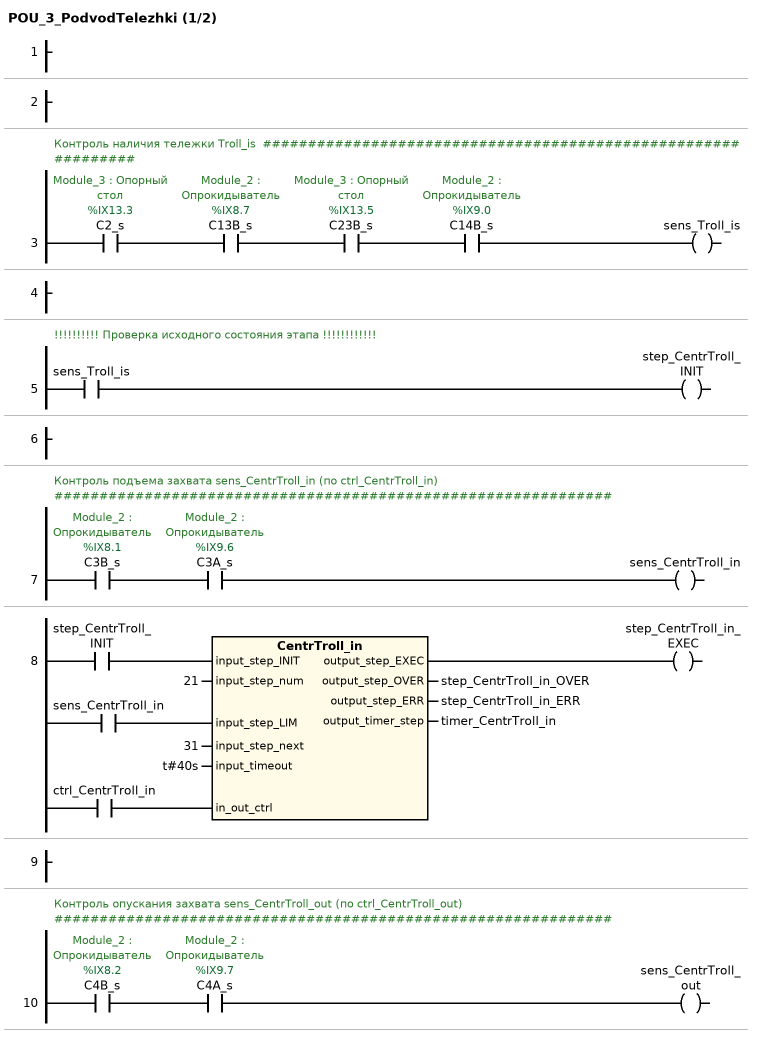
// NETWORK 1

// NETWORK 2

// NETWORK 3
// Контроль наличия тележки Troll_is  ##############################################################
//   C2_s: Module_3 : Опорный стол | AT %IX13.3
//   C13B_s: Module_2 : Опрокидыватель | AT %IX8.7
//   C23B_s: Module_3 : Опорный стол | AT %IX13.5
//   C14B_s: Module_2 : Опрокидыватель | AT %IX9.0
sens_Troll_is := C2_s AND C13B_s AND C23B_s AND C14B_s;

// NETWORK 4

// NETWORK 5
// !!!!!!!!!! Проверка исходного состояния этапа !!!!!!!!!!!!
step_CentrTroll_INIT := sens_Troll_is;

// NETWORK 6

// NETWORK 7
// Контроль подъема захвата sens_CentrTroll_in (по ctrl_CentrTroll_in) ##############################################################
//   C3B_s: Module_2 : Опрокидыватель | AT %IX8.1
//   C3A_s: Module_2 : Опрокидыватель | AT %IX9.6
sens_CentrTroll_in := C3B_s AND C3A_s;

// NETWORK 8
CentrTroll_in(input_step_INIT := step_CentrTroll_INIT, input_step_num := 21, input_step_LIM := sens_CentrTroll_in, input_step_next := 31, input_timeout := t#40s, in_out_ctrl := ctrl_CentrTroll_in, output_step_OVER => step_CentrTroll_in_OVER, output_step_ERR => step_CentrTroll_in_ERR, output_timer_step => timer_CentrTroll_in);
step_CentrTroll_in_EXEC := CentrTroll_in.output_step_EXEC;

// NETWORK 9

// NETWORK 10
// Контроль опускания захвата sens_CentrTroll_out (по ctrl_CentrTroll_out) ##############################################################
//   C4B_s: Module_2 : Опрокидыватель | AT %IX8.2
//   C4A_s: Module_2 : Опрокидыватель | AT %IX9.7
sens_CentrTroll_out := C4B_s AND C4A_s;

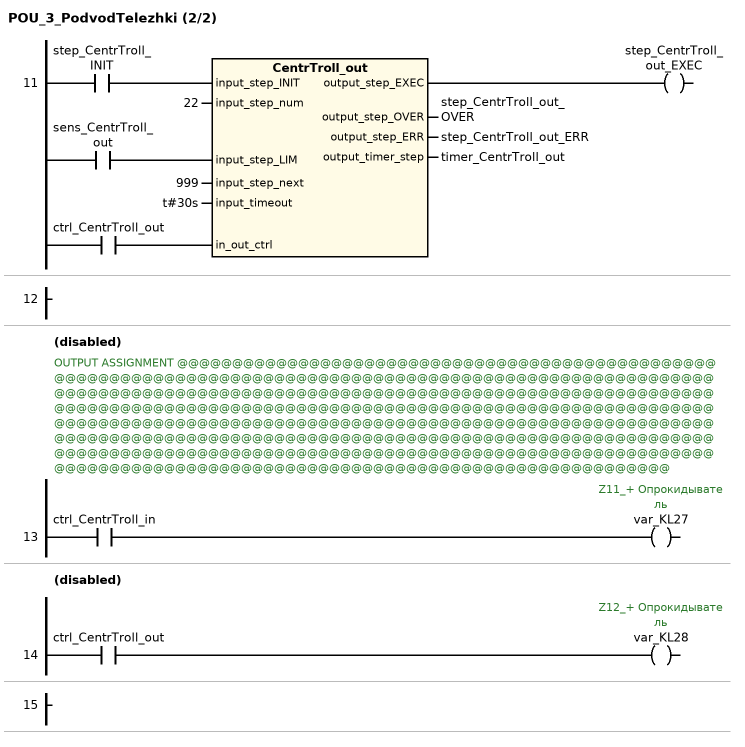
// NETWORK 11
CentrTroll_out(input_step_INIT := step_CentrTroll_INIT, input_step_num := 22, input_step_LIM := sens_CentrTroll_out, input_step_next := 999, input_timeout := t#30s, in_out_ctrl := ctrl_CentrTroll_out, output_step_OVER => step_CentrTroll_out_OVER, output_step_ERR => step_CentrTroll_out_ERR, output_timer_step => timer_CentrTroll_out);
step_CentrTroll_out_EXEC := CentrTroll_out.output_step_EXEC;

// NETWORK 12

// NETWORK 13 (disabled)
// OUTPUT ASSIGNMENT @@@@@@@@@@@@@@@@@@@@@@@@@@@@@@@@@@@@@@@@@@@@@@@@@@@@@@@@@@@@@@@@@@@@@@@@@@@@@@@@@@@@@@@@@@@@@@@@@@@@@@@@@@@@@@@@@@@@@@@@@@@@@@@@@@@@@@@@@@@@@@@@@@@@@@@@@@@@@@@@@@@@@@@@@@@@@@@@@@@@@@@@@@@@@@@@@@@@@@@@@@@@@@@@@@@@@@@@@@@@@@@@@@@@@@@@@@@@@@@@@@@@@@@@@@@@@@@@@@@@@@@@@@@@@@@@@@@@@@@@@@@@@@@@@@@@@@@@@@@@@@@@@@@@@@@@@@@@@@@@@@@@@@@@@@@@@@@@@@@@@@@@@@@@@@@@@@@@@@@@@@@@@@@@@@@@@@@@@@@@@@@@@@@@@@@@@@@@@@@@@@@@@@@@@@@@@@@@@@@@@@@@@@@@@@@@@@@@@@@@@@@@@@@@@@@@@@@@@@@@@@@@@
//   var_KL27: Z11_+ Опрокидыватель
// var_KL27 := ctrl_CentrTroll_in;

// NETWORK 14 (disabled)
//   var_KL28: Z12_+ Опрокидыватель
// var_KL28 := ctrl_CentrTroll_out;

// NETWORK 15

END_PROGRAM

// MyController/Application/module_unites/CentrTroll_in
PROGRAM CentrTroll_in
VAR_INPUT
	input_step_INIT: BOOL;
	input_step_num: INT;
	input_step_LIM: BOOL;
	input_step_next: INT;
	input_timeout: TIME;
END_VAR

VAR_OUTPUT
	output_step_EXEC: BOOL;
	output_step_OVER: BOOL;
	output_step_ERR: BOOL;
	output_timer_step: TIME;
END_VAR
VAR_IN_OUT
	in_out_ctrl: BOOL;
END_VAR
VAR
	TON_step: TON;
	TON_step_res: BOOL;
	step_active: BOOL;
	TON_delay: TON;
	timer_delay: TIME;
	ton_delay_ok: BOOL;
END_VAR
VAR // added by the converter: edge detectors and wires of the graphical bodies
    _rt1, _rt2, _rt3, _rt4, _rt5, _rt6, _rt7 : R_TRIG;
    _w1, _w2 : BOOL;
    _ft1 : F_TRIG;
END_VAR

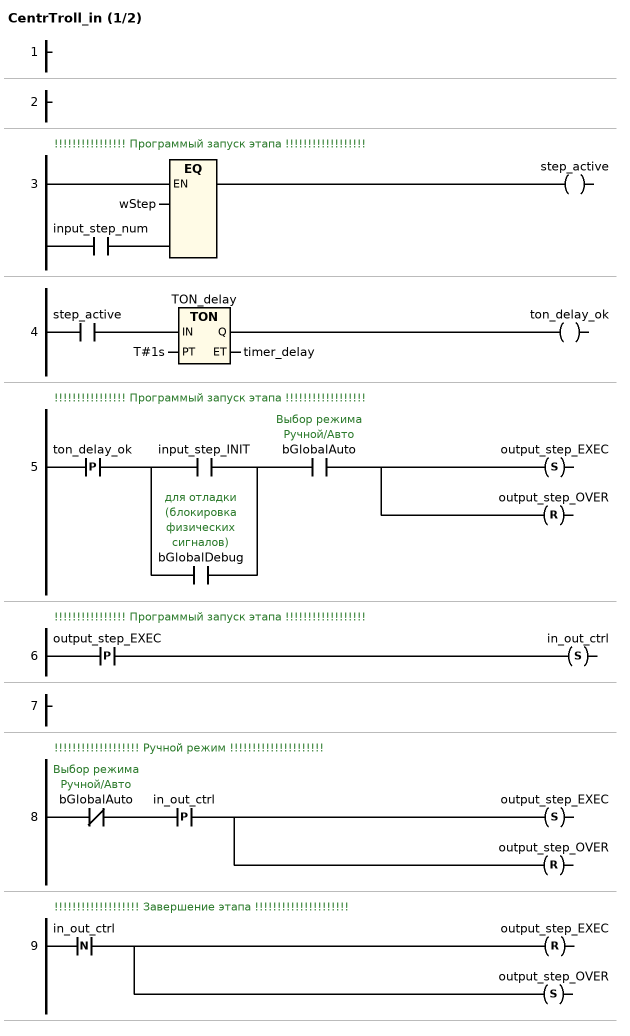
// NETWORK 1

// NETWORK 2

// NETWORK 3
// !!!!!!!!!!!!!!!! Программый запуск этапа !!!!!!!!!!!!!!!!!!
step_active := wStep = input_step_num;

// NETWORK 4
TON_delay(IN := step_active, PT := T#1s, ET => timer_delay); // TON
ton_delay_ok := TON_delay.Q;

// NETWORK 5
// !!!!!!!!!!!!!!!! Программый запуск этапа !!!!!!!!!!!!!!!!!!
//   bGlobalDebug: для отладки (блокировка физических сигналов)
//   bGlobalAuto: Выбор режима Ручной/Авто
_rt1(CLK := ton_delay_ok);
_w1 := _rt1.Q AND (input_step_INIT OR bGlobalDebug) AND bGlobalAuto;
output_step_EXEC S= _w1;
output_step_OVER R= _w1;

// NETWORK 6
// !!!!!!!!!!!!!!!! Программый запуск этапа !!!!!!!!!!!!!!!!!!
_rt2(CLK := output_step_EXEC);
in_out_ctrl S= _rt2.Q;

// NETWORK 7

// NETWORK 8
// !!!!!!!!!!!!!!!!!!! Ручной режим !!!!!!!!!!!!!!!!!!!!!
//   bGlobalAuto: Выбор режима Ручной/Авто
_rt3(CLK := in_out_ctrl);
_w2 := NOT bGlobalAuto AND _rt3.Q;
output_step_EXEC S= _w2;
output_step_OVER R= _w2;

// NETWORK 9
// !!!!!!!!!!!!!!!!!!! Завершение этапа !!!!!!!!!!!!!!!!!!!!!
_ft1(CLK := in_out_ctrl);
output_step_EXEC R= _ft1.Q;
output_step_OVER S= _ft1.Q;

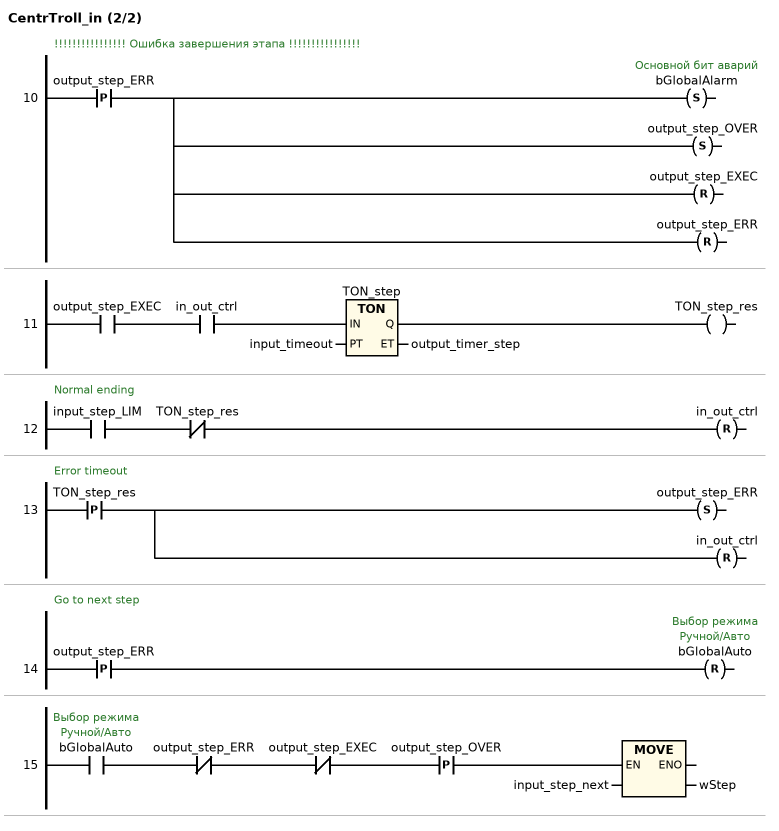
// NETWORK 10
// !!!!!!!!!!!!!!!! Ошибка завершения этапа !!!!!!!!!!!!!!!!
//   bGlobalAlarm: Основной бит аварий
_rt4(CLK := output_step_ERR);
bGlobalAlarm S= _rt4.Q;
output_step_OVER S= _rt4.Q;
output_step_EXEC R= _rt4.Q;
output_step_ERR R= _rt4.Q;

// NETWORK 11
TON_step(IN := output_step_EXEC AND in_out_ctrl, PT := input_timeout, ET => output_timer_step); // TON
TON_step_res := TON_step.Q;

// NETWORK 12
// Normal ending
in_out_ctrl R= input_step_LIM AND NOT TON_step_res;

// NETWORK 13
// Error timeout
_rt5(CLK := TON_step_res);
output_step_ERR S= _rt5.Q;
in_out_ctrl R= _rt5.Q;

// NETWORK 14
// Go to next step
//   bGlobalAuto: Выбор режима Ручной/Авто
_rt6(CLK := output_step_ERR);
bGlobalAuto R= _rt6.Q;

// NETWORK 15
//   bGlobalAuto: Выбор режима Ручной/Авто
_rt7(CLK := output_step_OVER);
IF bGlobalAuto AND NOT output_step_ERR AND NOT output_step_EXEC AND _rt7.Q THEN wStep := input_step_next; END_IF

END_PROGRAM

// MyController/Application/module_unites/CentrTroll_out
PROGRAM CentrTroll_out
VAR_INPUT
	input_step_INIT: BOOL;
	input_step_num: INT;
	input_step_LIM: BOOL;
	input_step_next: INT;
	input_timeout: TIME;
END_VAR

VAR_OUTPUT
	output_step_EXEC: BOOL;
	output_step_OVER: BOOL;
	output_step_ERR: BOOL;
	output_timer_step: TIME;
END_VAR
VAR_IN_OUT
	in_out_ctrl: BOOL;
END_VAR
VAR
	TON_step: TON;
	TON_step_res: BOOL;
	step_active: BOOL;
	TON_delay: TON;
	timer_delay: TIME;
	ton_delay_ok: BOOL;
END_VAR
VAR // added by the converter: edge detectors and wires of the graphical bodies
    _rt1, _rt2, _rt3, _rt4, _rt5, _rt6, _rt7 : R_TRIG;
    _w1, _w2 : BOOL;
    _ft1 : F_TRIG;
END_VAR

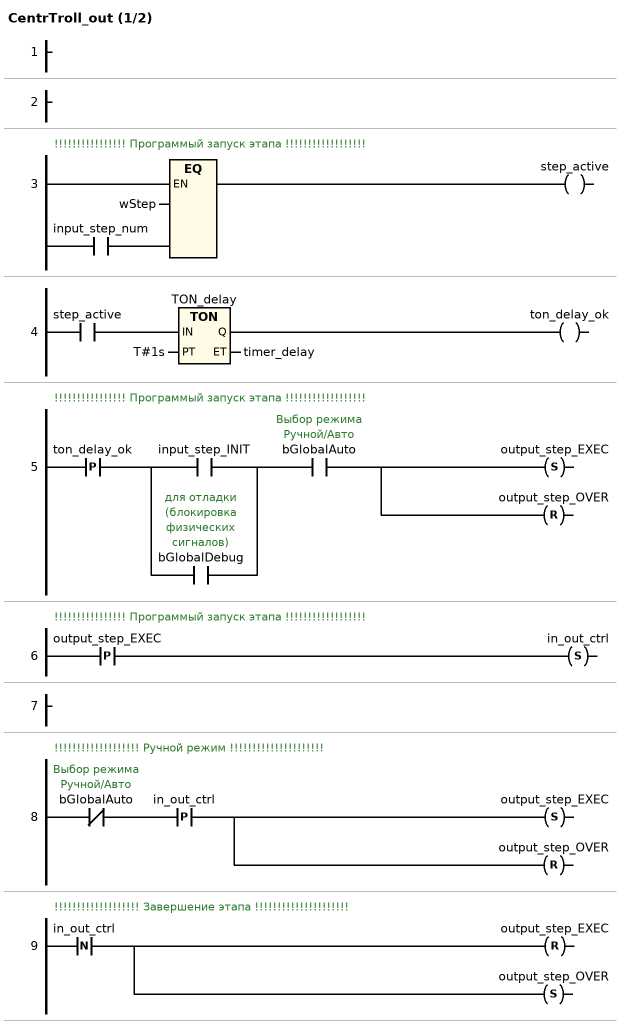
// NETWORK 1

// NETWORK 2

// NETWORK 3
// !!!!!!!!!!!!!!!! Программый запуск этапа !!!!!!!!!!!!!!!!!!
step_active := wStep = input_step_num;

// NETWORK 4
TON_delay(IN := step_active, PT := T#1s, ET => timer_delay); // TON
ton_delay_ok := TON_delay.Q;

// NETWORK 5
// !!!!!!!!!!!!!!!! Программый запуск этапа !!!!!!!!!!!!!!!!!!
//   bGlobalDebug: для отладки (блокировка физических сигналов)
//   bGlobalAuto: Выбор режима Ручной/Авто
_rt1(CLK := ton_delay_ok);
_w1 := _rt1.Q AND (input_step_INIT OR bGlobalDebug) AND bGlobalAuto;
output_step_EXEC S= _w1;
output_step_OVER R= _w1;

// NETWORK 6
// !!!!!!!!!!!!!!!! Программый запуск этапа !!!!!!!!!!!!!!!!!!
_rt2(CLK := output_step_EXEC);
in_out_ctrl S= _rt2.Q;

// NETWORK 7

// NETWORK 8
// !!!!!!!!!!!!!!!!!!! Ручной режим !!!!!!!!!!!!!!!!!!!!!
//   bGlobalAuto: Выбор режима Ручной/Авто
_rt3(CLK := in_out_ctrl);
_w2 := NOT bGlobalAuto AND _rt3.Q;
output_step_EXEC S= _w2;
output_step_OVER R= _w2;

// NETWORK 9
// !!!!!!!!!!!!!!!!!!! Завершение этапа !!!!!!!!!!!!!!!!!!!!!
_ft1(CLK := in_out_ctrl);
output_step_EXEC R= _ft1.Q;
output_step_OVER S= _ft1.Q;

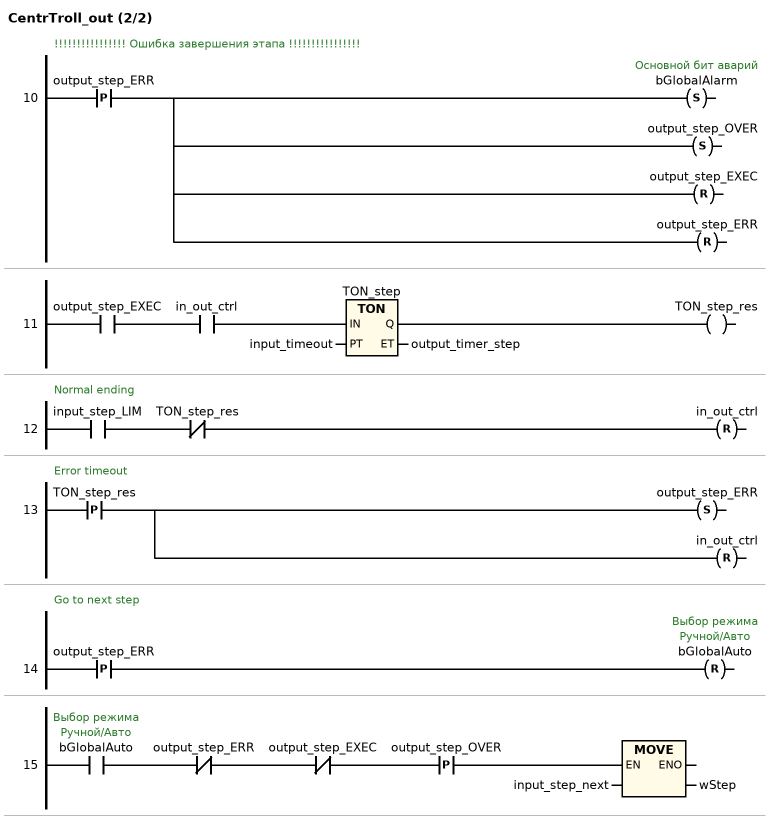
// NETWORK 10
// !!!!!!!!!!!!!!!! Ошибка завершения этапа !!!!!!!!!!!!!!!!
//   bGlobalAlarm: Основной бит аварий
_rt4(CLK := output_step_ERR);
bGlobalAlarm S= _rt4.Q;
output_step_OVER S= _rt4.Q;
output_step_EXEC R= _rt4.Q;
output_step_ERR R= _rt4.Q;

// NETWORK 11
TON_step(IN := output_step_EXEC AND in_out_ctrl, PT := input_timeout, ET => output_timer_step); // TON
TON_step_res := TON_step.Q;

// NETWORK 12
// Normal ending
in_out_ctrl R= input_step_LIM AND NOT TON_step_res;

// NETWORK 13
// Error timeout
_rt5(CLK := TON_step_res);
output_step_ERR S= _rt5.Q;
in_out_ctrl R= _rt5.Q;

// NETWORK 14
// Go to next step
//   bGlobalAuto: Выбор режима Ручной/Авто
_rt6(CLK := output_step_ERR);
bGlobalAuto R= _rt6.Q;

// NETWORK 15
//   bGlobalAuto: Выбор режима Ручной/Авто
_rt7(CLK := output_step_OVER);
IF bGlobalAuto AND NOT output_step_ERR AND NOT output_step_EXEC AND _rt7.Q THEN wStep := input_step_next; END_IF

END_PROGRAM

// MyController/Application/POU_4_Zahvat
PROGRAM POU_4_Zahvat
VAR
	timer_GrabTroll_in: TIME;
	sens_GrabTroll_in: BOOL;
	ctrl_GrabTroll_in: BOOL;
	timer_GrabTroll_out: TIME;
	sens_GrabTroll_out: BOOL;
	ctrl_GrabTroll_out: BOOL;
	timer_TurnTroll_in: TIME;
	sens_TurnTroll_in: BOOL;
	ctrl_TurnTroll_in: BOOL;
	timer_TurnTroll_out: TIME;
	sens_TurnTroll_out: BOOL;
	ctrl_TurnTroll_out: BOOL;
	step_GrabTroll_in_OVER: BOOL;
	step_GrabTroll_in_ERR: BOOL;
	step_GrabTroll_in_EXEC: BOOL;
	step_GrabTroll_INIT: BOOL := TRUE;
	step_GrabTroll_out_OVER: BOOL;
	step_GrabTroll_out_ERR: BOOL;
	step_GrabTroll_out_EXEC: BOOL;
	step_TurnTroll_INIT: BOOL := TRUE;
	step_TurnTroll_out_EXEC: BOOL;
	step_TurnTroll_in_EXEC: BOOL;
	step_TurnTroll_in_OVER: BOOL;
	step_TurnTroll_in_ERR: BOOL;
	step_TurnTroll_out_OVER: BOOL;
	step_TurnTroll_out_ERR: BOOL;
END_VAR

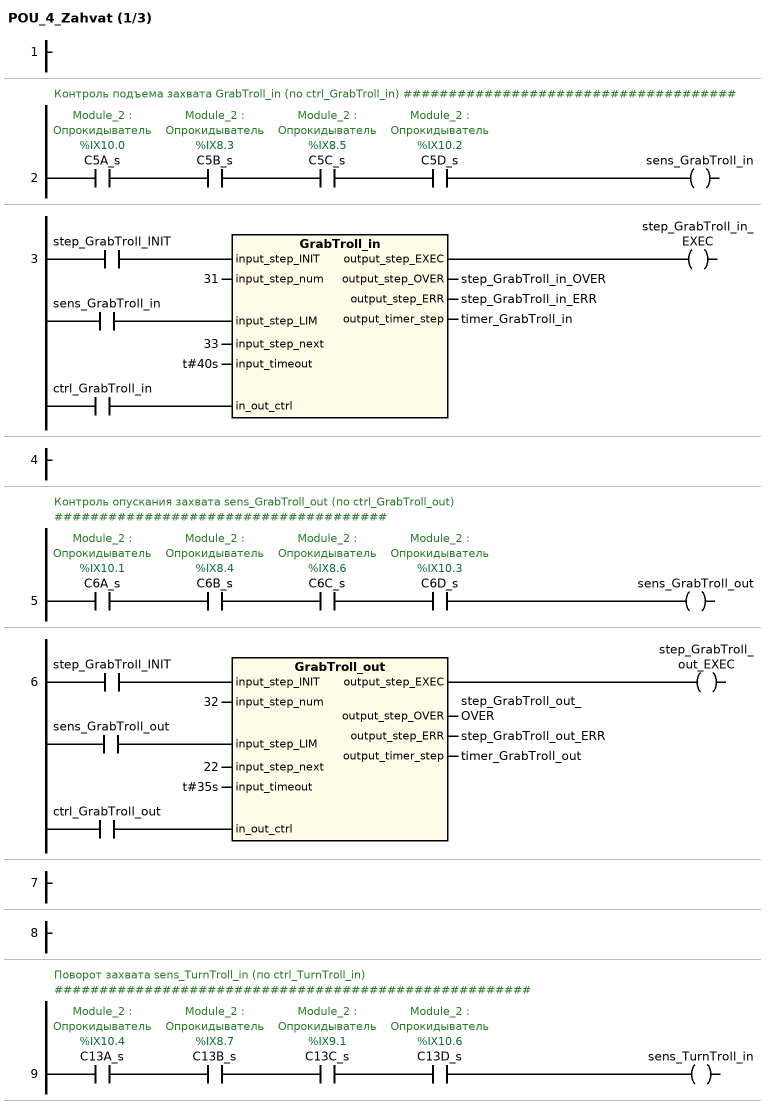
// NETWORK 1

// NETWORK 2
// Контроль подъема захвата GrabTroll_in (по ctrl_GrabTroll_in) #####################################
//   C5A_s: Module_2 : Опрокидыватель | AT %IX10.0
//   C5B_s: Module_2 : Опрокидыватель | AT %IX8.3
//   C5C_s: Module_2 : Опрокидыватель | AT %IX8.5
//   C5D_s: Module_2 : Опрокидыватель | AT %IX10.2
sens_GrabTroll_in := C5A_s AND C5B_s AND C5C_s AND C5D_s;

// NETWORK 3
GrabTroll_in(input_step_INIT := step_GrabTroll_INIT, input_step_num := 31, input_step_LIM := sens_GrabTroll_in, input_step_next := 33, input_timeout := t#40s, in_out_ctrl := ctrl_GrabTroll_in, output_step_OVER => step_GrabTroll_in_OVER, output_step_ERR => step_GrabTroll_in_ERR, output_timer_step => timer_GrabTroll_in);
step_GrabTroll_in_EXEC := GrabTroll_in.output_step_EXEC;

// NETWORK 4

// NETWORK 5
// Контроль опускания захвата sens_GrabTroll_out (по ctrl_GrabTroll_out) #####################################
//   C6A_s: Module_2 : Опрокидыватель | AT %IX10.1
//   C6B_s: Module_2 : Опрокидыватель | AT %IX8.4
//   C6C_s: Module_2 : Опрокидыватель | AT %IX8.6
//   C6D_s: Module_2 : Опрокидыватель | AT %IX10.3
sens_GrabTroll_out := C6A_s AND C6B_s AND C6C_s AND C6D_s;

// NETWORK 6
GrabTroll_out(input_step_INIT := step_GrabTroll_INIT, input_step_num := 32, input_step_LIM := sens_GrabTroll_out, input_step_next := 22, input_timeout := t#35s, in_out_ctrl := ctrl_GrabTroll_out, output_step_OVER => step_GrabTroll_out_OVER, output_step_ERR => step_GrabTroll_out_ERR, output_timer_step => timer_GrabTroll_out);
step_GrabTroll_out_EXEC := GrabTroll_out.output_step_EXEC;

// NETWORK 7

// NETWORK 8

// NETWORK 9
// Поворот захвата sens_TurnTroll_in (по ctrl_TurnTroll_in) #####################################################
//   C13A_s: Module_2 : Опрокидыватель | AT %IX10.4
//   C13B_s: Module_2 : Опрокидыватель | AT %IX8.7
//   C13C_s: Module_2 : Опрокидыватель | AT %IX9.1
//   C13D_s: Module_2 : Опрокидыватель | AT %IX10.6
sens_TurnTroll_in := C13A_s AND C13B_s AND C13C_s AND C13D_s;

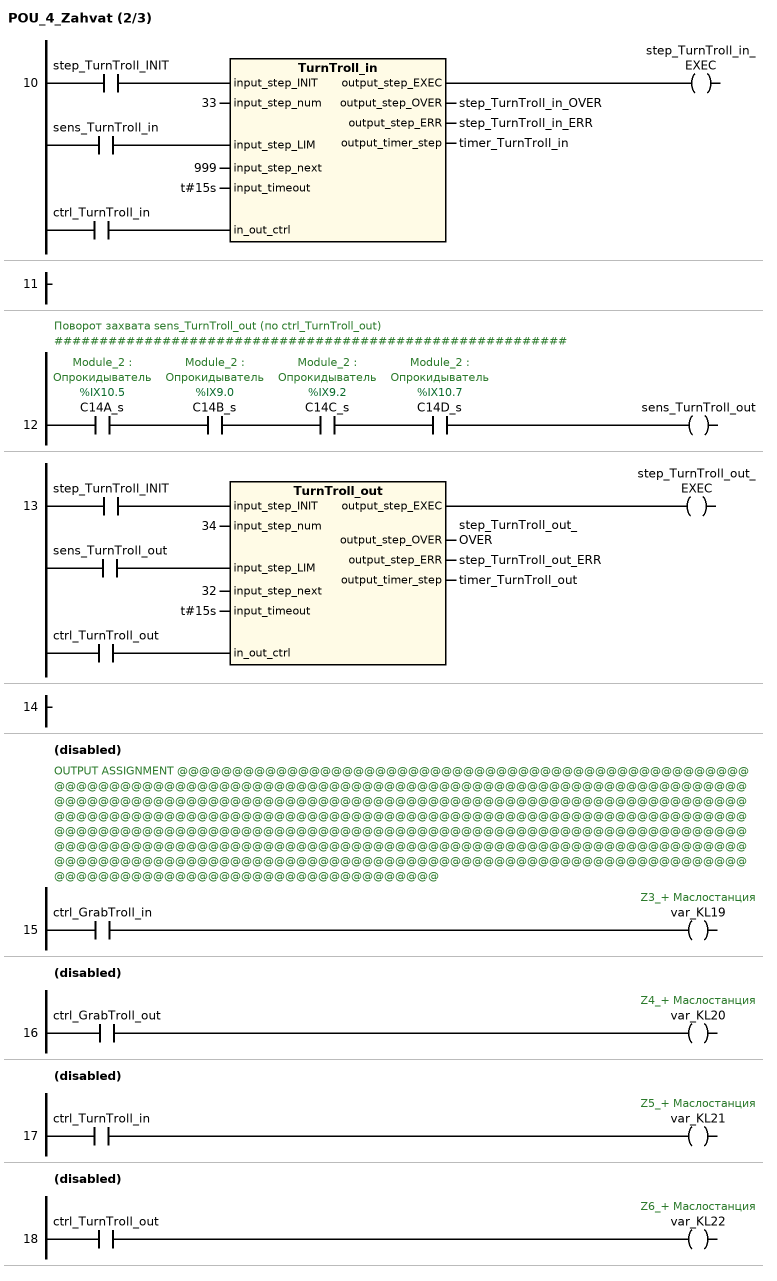
// NETWORK 10
TurnTroll_in(input_step_INIT := step_TurnTroll_INIT, input_step_num := 33, input_step_LIM := sens_TurnTroll_in, input_step_next := 999, input_timeout := t#15s, in_out_ctrl := ctrl_TurnTroll_in, output_step_OVER => step_TurnTroll_in_OVER, output_step_ERR => step_TurnTroll_in_ERR, output_timer_step => timer_TurnTroll_in);
step_TurnTroll_in_EXEC := TurnTroll_in.output_step_EXEC;

// NETWORK 11

// NETWORK 12
// Поворот захвата sens_TurnTroll_out (по ctrl_TurnTroll_out) #########################################################
//   C14A_s: Module_2 : Опрокидыватель | AT %IX10.5
//   C14B_s: Module_2 : Опрокидыватель | AT %IX9.0
//   C14C_s: Module_2 : Опрокидыватель | AT %IX9.2
//   C14D_s: Module_2 : Опрокидыватель | AT %IX10.7
sens_TurnTroll_out := C14A_s AND C14B_s AND C14C_s AND C14D_s;

// NETWORK 13
TurnTroll_out(input_step_INIT := step_TurnTroll_INIT, input_step_num := 34, input_step_LIM := sens_TurnTroll_out, input_step_next := 32, input_timeout := t#15s, in_out_ctrl := ctrl_TurnTroll_out, output_step_OVER => step_TurnTroll_out_OVER, output_step_ERR => step_TurnTroll_out_ERR, output_timer_step => timer_TurnTroll_out);
step_TurnTroll_out_EXEC := TurnTroll_out.output_step_EXEC;

// NETWORK 14

// NETWORK 15 (disabled)
// OUTPUT ASSIGNMENT @@@@@@@@@@@@@@@@@@@@@@@@@@@@@@@@@@@@@@@@@@@@@@@@@@@@@@@@@@@@@@@@@@@@@@@@@@@@@@@@@@@@@@@@@@@@@@@@@@@@@@@@@@@@@@@@@@@@@@@@@@@@@@@@@@@@@@@@@@@@@@@@@@@@@@@@@@@@@@@@@@@@@@@@@@@@@@@@@@@@@@@@@@@@@@@@@@@@@@@@@@@@@@@@@@@@@@@@@@@@@@@@@@@@@@@@@@@@@@@@@@@@@@@@@@@@@@@@@@@@@@@@@@@@@@@@@@@@@@@@@@@@@@@@@@@@@@@@@@@@@@@@@@@@@@@@@@@@@@@@@@@@@@@@@@@@@@@@@@@@@@@@@@@@@@@@@@@@@@@@@@@@@@@@@@@@@@@@@@@@@@@@@@@@@@@@@@@@@@@@@@@@@@@@@@@@@@@@@@@@@@@@@@@@@@@@@@@@@@@@@@@@@@@@@@@@@@@@@@@@@@@@@
//   var_KL19: Z3_+ Маслостанция
// var_KL19 := ctrl_GrabTroll_in;

// NETWORK 16 (disabled)
//   var_KL20: Z4_+ Маслостанция
// var_KL20 := ctrl_GrabTroll_out;

// NETWORK 17 (disabled)
//   var_KL21: Z5_+ Маслостанция
// var_KL21 := ctrl_TurnTroll_in;

// NETWORK 18 (disabled)
//   var_KL22: Z6_+ Маслостанция
// var_KL22 := ctrl_TurnTroll_out;

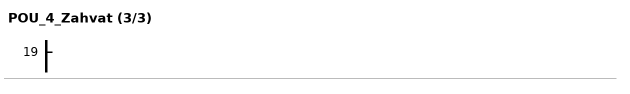
// NETWORK 19

END_PROGRAM

// MyController/Application/module_unites/GrabTroll_in
PROGRAM GrabTroll_in
VAR_INPUT
	input_step_INIT: BOOL;
	input_step_num: INT;
	input_step_LIM: BOOL;
	input_step_next: INT;
	input_timeout: TIME;
END_VAR

VAR_OUTPUT
	output_step_EXEC: BOOL;
	output_step_OVER: BOOL;
	output_step_ERR: BOOL;
	output_timer_step: TIME;
END_VAR
VAR_IN_OUT
	in_out_ctrl: BOOL;
END_VAR
VAR
	TON_step: TON;
	TON_step_res: BOOL;
	step_active: BOOL;
	TON_delay: TON;
	timer_delay: TIME;
	ton_delay_ok: BOOL;
END_VAR
VAR // added by the converter: edge detectors and wires of the graphical bodies
    _rt1, _rt2, _rt3, _rt4, _rt5, _rt6, _rt7 : R_TRIG;
    _w1, _w2 : BOOL;
    _ft1 : F_TRIG;
END_VAR

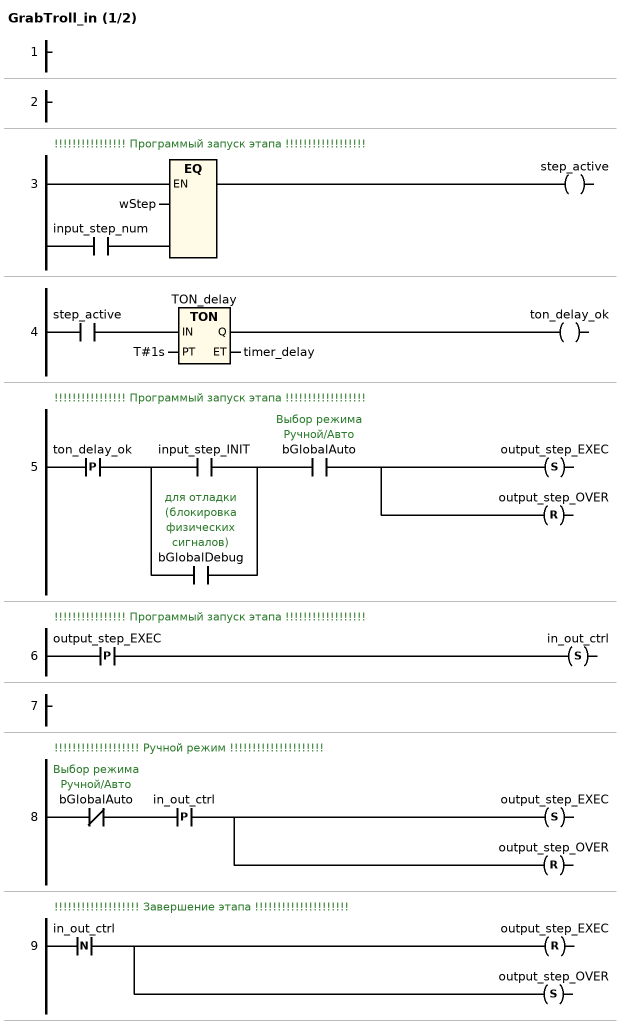
// NETWORK 1

// NETWORK 2

// NETWORK 3
// !!!!!!!!!!!!!!!! Программый запуск этапа !!!!!!!!!!!!!!!!!!
step_active := wStep = input_step_num;

// NETWORK 4
TON_delay(IN := step_active, PT := T#1s, ET => timer_delay); // TON
ton_delay_ok := TON_delay.Q;

// NETWORK 5
// !!!!!!!!!!!!!!!! Программый запуск этапа !!!!!!!!!!!!!!!!!!
//   bGlobalDebug: для отладки (блокировка физических сигналов)
//   bGlobalAuto: Выбор режима Ручной/Авто
_rt1(CLK := ton_delay_ok);
_w1 := _rt1.Q AND (input_step_INIT OR bGlobalDebug) AND bGlobalAuto;
output_step_EXEC S= _w1;
output_step_OVER R= _w1;

// NETWORK 6
// !!!!!!!!!!!!!!!! Программый запуск этапа !!!!!!!!!!!!!!!!!!
_rt2(CLK := output_step_EXEC);
in_out_ctrl S= _rt2.Q;

// NETWORK 7

// NETWORK 8
// !!!!!!!!!!!!!!!!!!! Ручной режим !!!!!!!!!!!!!!!!!!!!!
//   bGlobalAuto: Выбор режима Ручной/Авто
_rt3(CLK := in_out_ctrl);
_w2 := NOT bGlobalAuto AND _rt3.Q;
output_step_EXEC S= _w2;
output_step_OVER R= _w2;

// NETWORK 9
// !!!!!!!!!!!!!!!!!!! Завершение этапа !!!!!!!!!!!!!!!!!!!!!
_ft1(CLK := in_out_ctrl);
output_step_EXEC R= _ft1.Q;
output_step_OVER S= _ft1.Q;

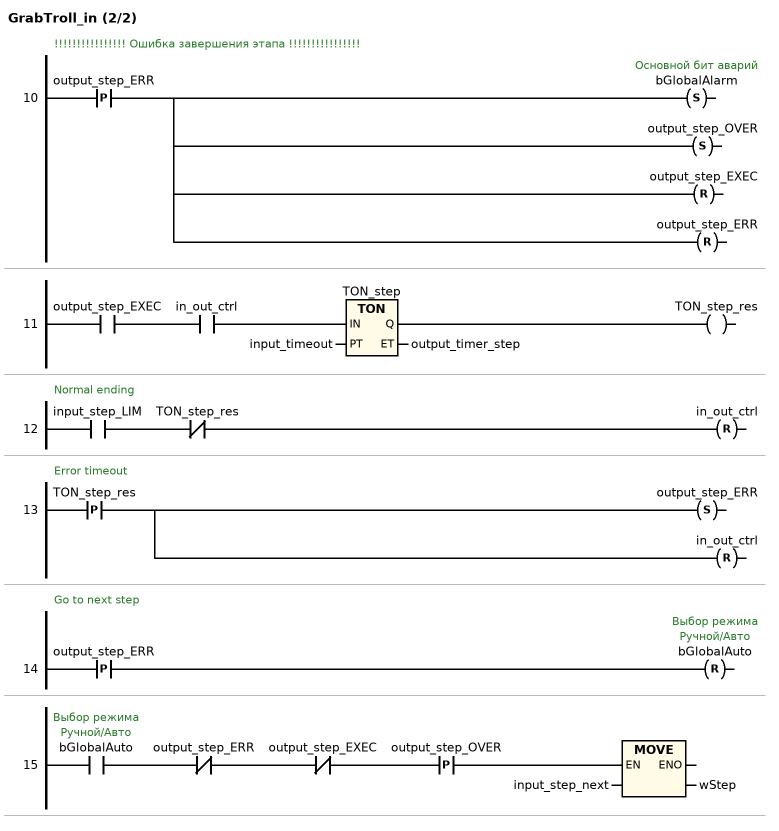
// NETWORK 10
// !!!!!!!!!!!!!!!! Ошибка завершения этапа !!!!!!!!!!!!!!!!
//   bGlobalAlarm: Основной бит аварий
_rt4(CLK := output_step_ERR);
bGlobalAlarm S= _rt4.Q;
output_step_OVER S= _rt4.Q;
output_step_EXEC R= _rt4.Q;
output_step_ERR R= _rt4.Q;

// NETWORK 11
TON_step(IN := output_step_EXEC AND in_out_ctrl, PT := input_timeout, ET => output_timer_step); // TON
TON_step_res := TON_step.Q;

// NETWORK 12
// Normal ending
in_out_ctrl R= input_step_LIM AND NOT TON_step_res;

// NETWORK 13
// Error timeout
_rt5(CLK := TON_step_res);
output_step_ERR S= _rt5.Q;
in_out_ctrl R= _rt5.Q;

// NETWORK 14
// Go to next step
//   bGlobalAuto: Выбор режима Ручной/Авто
_rt6(CLK := output_step_ERR);
bGlobalAuto R= _rt6.Q;

// NETWORK 15
//   bGlobalAuto: Выбор режима Ручной/Авто
_rt7(CLK := output_step_OVER);
IF bGlobalAuto AND NOT output_step_ERR AND NOT output_step_EXEC AND _rt7.Q THEN wStep := input_step_next; END_IF

END_PROGRAM

// MyController/Application/module_unites/GrabTroll_out
PROGRAM GrabTroll_out
VAR_INPUT
	input_step_INIT: BOOL;
	input_step_num: INT;
	input_step_LIM: BOOL;
	input_step_next: INT;
	input_timeout: TIME;
END_VAR

VAR_OUTPUT
	output_step_EXEC: BOOL;
	output_step_OVER: BOOL;
	output_step_ERR: BOOL;
	output_timer_step: TIME;
END_VAR
VAR_IN_OUT
	in_out_ctrl: BOOL;
END_VAR
VAR
	TON_step: TON;
	TON_step_res: BOOL;
	step_active: BOOL;
	TON_delay: TON;
	timer_delay: TIME;
	ton_delay_ok: BOOL;
END_VAR
VAR // added by the converter: edge detectors and wires of the graphical bodies
    _rt1, _rt2, _rt3, _rt4, _rt5, _rt6, _rt7 : R_TRIG;
    _w1, _w2 : BOOL;
    _ft1 : F_TRIG;
END_VAR

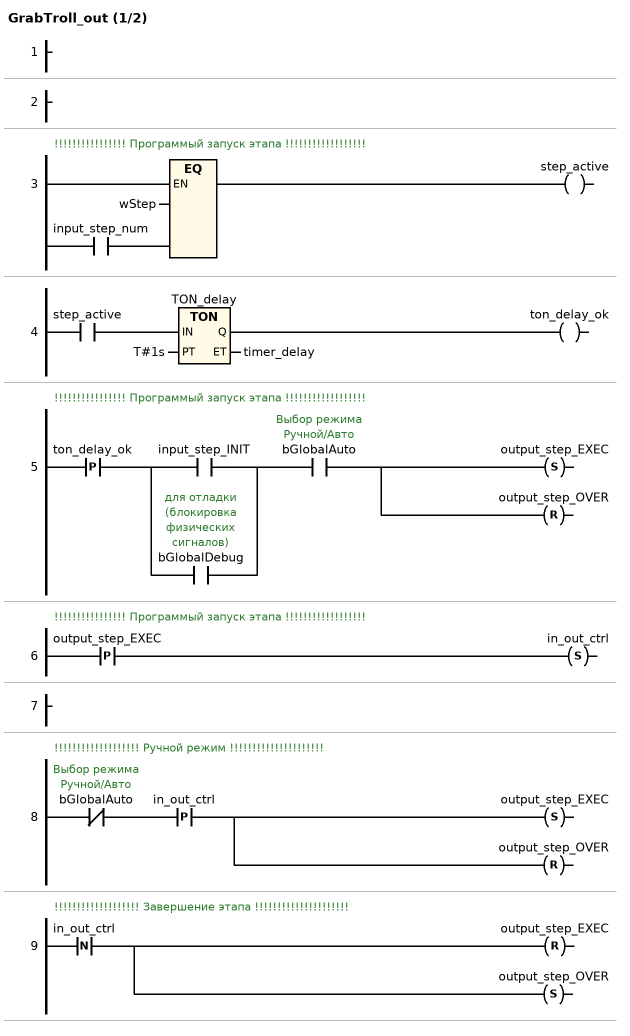
// NETWORK 1

// NETWORK 2

// NETWORK 3
// !!!!!!!!!!!!!!!! Программый запуск этапа !!!!!!!!!!!!!!!!!!
step_active := wStep = input_step_num;

// NETWORK 4
TON_delay(IN := step_active, PT := T#1s, ET => timer_delay); // TON
ton_delay_ok := TON_delay.Q;

// NETWORK 5
// !!!!!!!!!!!!!!!! Программый запуск этапа !!!!!!!!!!!!!!!!!!
//   bGlobalDebug: для отладки (блокировка физических сигналов)
//   bGlobalAuto: Выбор режима Ручной/Авто
_rt1(CLK := ton_delay_ok);
_w1 := _rt1.Q AND (input_step_INIT OR bGlobalDebug) AND bGlobalAuto;
output_step_EXEC S= _w1;
output_step_OVER R= _w1;

// NETWORK 6
// !!!!!!!!!!!!!!!! Программый запуск этапа !!!!!!!!!!!!!!!!!!
_rt2(CLK := output_step_EXEC);
in_out_ctrl S= _rt2.Q;

// NETWORK 7

// NETWORK 8
// !!!!!!!!!!!!!!!!!!! Ручной режим !!!!!!!!!!!!!!!!!!!!!
//   bGlobalAuto: Выбор режима Ручной/Авто
_rt3(CLK := in_out_ctrl);
_w2 := NOT bGlobalAuto AND _rt3.Q;
output_step_EXEC S= _w2;
output_step_OVER R= _w2;

// NETWORK 9
// !!!!!!!!!!!!!!!!!!! Завершение этапа !!!!!!!!!!!!!!!!!!!!!
_ft1(CLK := in_out_ctrl);
output_step_EXEC R= _ft1.Q;
output_step_OVER S= _ft1.Q;

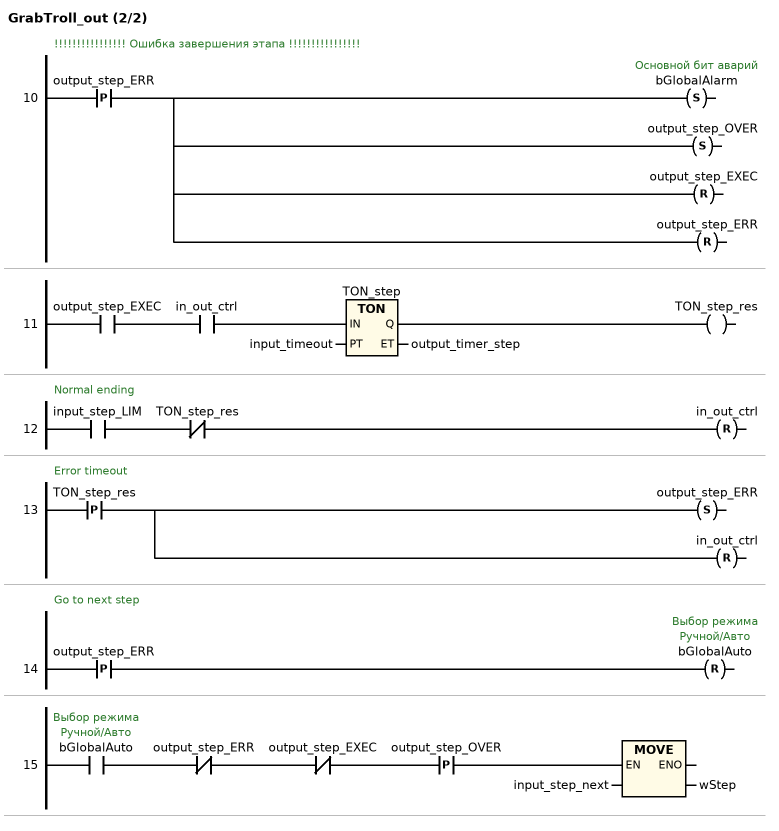
// NETWORK 10
// !!!!!!!!!!!!!!!! Ошибка завершения этапа !!!!!!!!!!!!!!!!
//   bGlobalAlarm: Основной бит аварий
_rt4(CLK := output_step_ERR);
bGlobalAlarm S= _rt4.Q;
output_step_OVER S= _rt4.Q;
output_step_EXEC R= _rt4.Q;
output_step_ERR R= _rt4.Q;

// NETWORK 11
TON_step(IN := output_step_EXEC AND in_out_ctrl, PT := input_timeout, ET => output_timer_step); // TON
TON_step_res := TON_step.Q;

// NETWORK 12
// Normal ending
in_out_ctrl R= input_step_LIM AND NOT TON_step_res;

// NETWORK 13
// Error timeout
_rt5(CLK := TON_step_res);
output_step_ERR S= _rt5.Q;
in_out_ctrl R= _rt5.Q;

// NETWORK 14
// Go to next step
//   bGlobalAuto: Выбор режима Ручной/Авто
_rt6(CLK := output_step_ERR);
bGlobalAuto R= _rt6.Q;

// NETWORK 15
//   bGlobalAuto: Выбор режима Ручной/Авто
_rt7(CLK := output_step_OVER);
IF bGlobalAuto AND NOT output_step_ERR AND NOT output_step_EXEC AND _rt7.Q THEN wStep := input_step_next; END_IF

END_PROGRAM

// MyController/Application/module_unites/TurnTroll_in
PROGRAM TurnTroll_in
VAR_INPUT
	input_step_INIT: BOOL;
	input_step_num: INT;
	input_step_LIM: BOOL;
	input_step_next: INT;
	input_timeout: TIME;
END_VAR

VAR_OUTPUT
	output_step_EXEC: BOOL;
	output_step_OVER: BOOL;
	output_step_ERR: BOOL;
	output_timer_step: TIME;
END_VAR
VAR_IN_OUT
	in_out_ctrl: BOOL;
END_VAR
VAR
	TON_step: TON;
	TON_step_res: BOOL;
	step_active: BOOL;
	TON_delay: TON;
	timer_delay: TIME;
	ton_delay_ok: BOOL;
END_VAR
VAR // added by the converter: edge detectors and wires of the graphical bodies
    _rt1, _rt2, _rt3, _rt4, _rt5, _rt6, _rt7 : R_TRIG;
    _w1, _w2 : BOOL;
    _ft1 : F_TRIG;
END_VAR

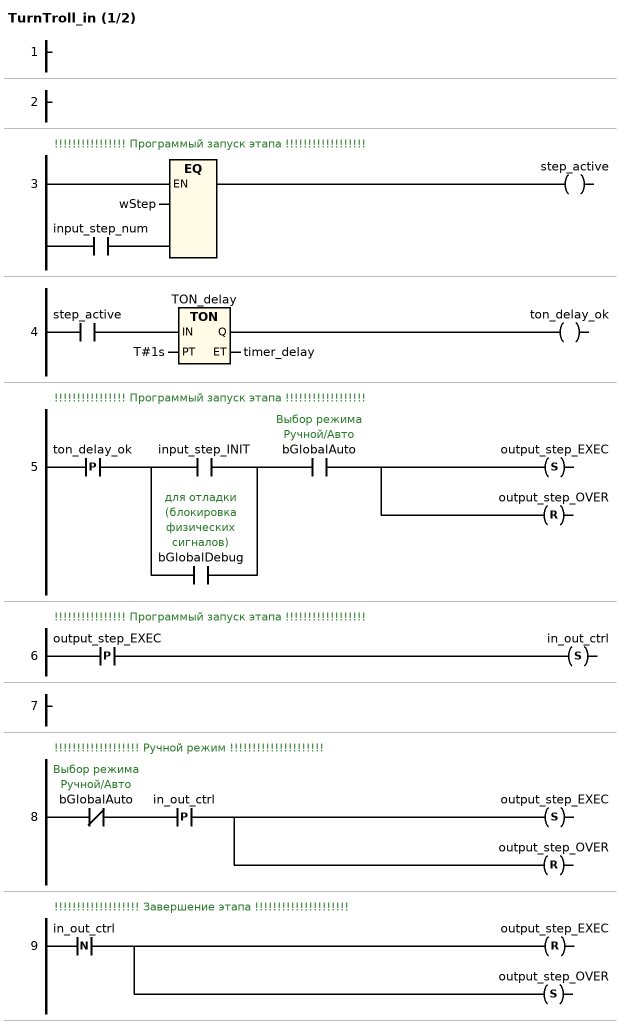
// NETWORK 1

// NETWORK 2

// NETWORK 3
// !!!!!!!!!!!!!!!! Программый запуск этапа !!!!!!!!!!!!!!!!!!
step_active := wStep = input_step_num;

// NETWORK 4
TON_delay(IN := step_active, PT := T#1s, ET => timer_delay); // TON
ton_delay_ok := TON_delay.Q;

// NETWORK 5
// !!!!!!!!!!!!!!!! Программый запуск этапа !!!!!!!!!!!!!!!!!!
//   bGlobalDebug: для отладки (блокировка физических сигналов)
//   bGlobalAuto: Выбор режима Ручной/Авто
_rt1(CLK := ton_delay_ok);
_w1 := _rt1.Q AND (input_step_INIT OR bGlobalDebug) AND bGlobalAuto;
output_step_EXEC S= _w1;
output_step_OVER R= _w1;

// NETWORK 6
// !!!!!!!!!!!!!!!! Программый запуск этапа !!!!!!!!!!!!!!!!!!
_rt2(CLK := output_step_EXEC);
in_out_ctrl S= _rt2.Q;

// NETWORK 7

// NETWORK 8
// !!!!!!!!!!!!!!!!!!! Ручной режим !!!!!!!!!!!!!!!!!!!!!
//   bGlobalAuto: Выбор режима Ручной/Авто
_rt3(CLK := in_out_ctrl);
_w2 := NOT bGlobalAuto AND _rt3.Q;
output_step_EXEC S= _w2;
output_step_OVER R= _w2;

// NETWORK 9
// !!!!!!!!!!!!!!!!!!! Завершение этапа !!!!!!!!!!!!!!!!!!!!!
_ft1(CLK := in_out_ctrl);
output_step_EXEC R= _ft1.Q;
output_step_OVER S= _ft1.Q;

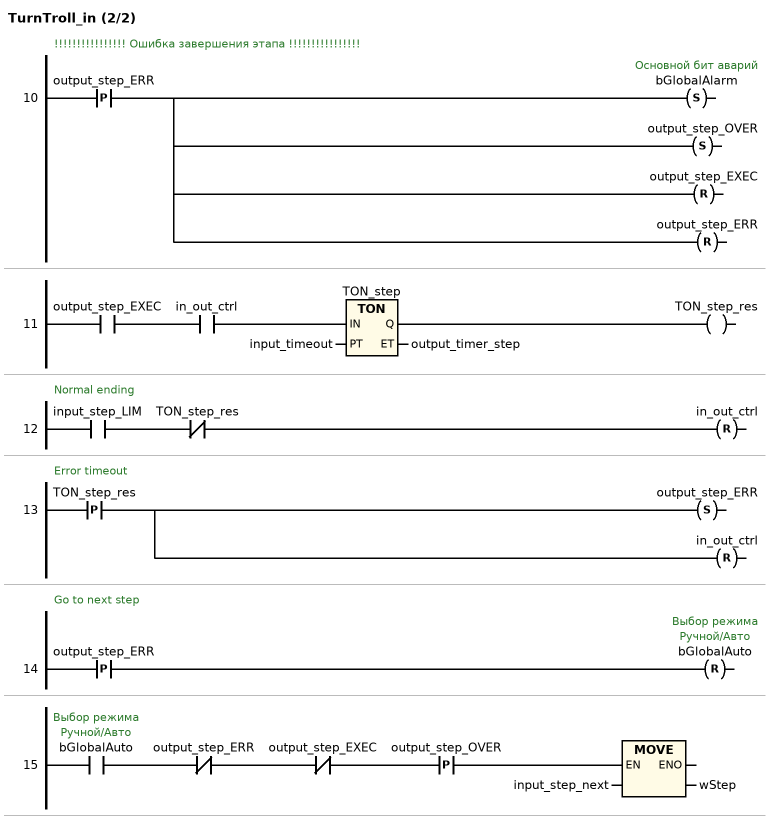
// NETWORK 10
// !!!!!!!!!!!!!!!! Ошибка завершения этапа !!!!!!!!!!!!!!!!
//   bGlobalAlarm: Основной бит аварий
_rt4(CLK := output_step_ERR);
bGlobalAlarm S= _rt4.Q;
output_step_OVER S= _rt4.Q;
output_step_EXEC R= _rt4.Q;
output_step_ERR R= _rt4.Q;

// NETWORK 11
TON_step(IN := output_step_EXEC AND in_out_ctrl, PT := input_timeout, ET => output_timer_step); // TON
TON_step_res := TON_step.Q;

// NETWORK 12
// Normal ending
in_out_ctrl R= input_step_LIM AND NOT TON_step_res;

// NETWORK 13
// Error timeout
_rt5(CLK := TON_step_res);
output_step_ERR S= _rt5.Q;
in_out_ctrl R= _rt5.Q;

// NETWORK 14
// Go to next step
//   bGlobalAuto: Выбор режима Ручной/Авто
_rt6(CLK := output_step_ERR);
bGlobalAuto R= _rt6.Q;

// NETWORK 15
//   bGlobalAuto: Выбор режима Ручной/Авто
_rt7(CLK := output_step_OVER);
IF bGlobalAuto AND NOT output_step_ERR AND NOT output_step_EXEC AND _rt7.Q THEN wStep := input_step_next; END_IF

END_PROGRAM

// MyController/Application/module_unites/TurnTroll_out
PROGRAM TurnTroll_out
VAR_INPUT
	input_step_INIT: BOOL;
	input_step_num: INT;
	input_step_LIM: BOOL;
	input_step_next: INT;
	input_timeout: TIME;
END_VAR

VAR_OUTPUT
	output_step_EXEC: BOOL;
	output_step_OVER: BOOL;
	output_step_ERR: BOOL;
	output_timer_step: TIME;
END_VAR
VAR_IN_OUT
	in_out_ctrl: BOOL;
END_VAR
VAR
	TON_step: TON;
	TON_step_res: BOOL;
	step_active: BOOL;
	TON_delay: TON;
	timer_delay: TIME;
	ton_delay_ok: BOOL;
END_VAR
VAR // added by the converter: edge detectors and wires of the graphical bodies
    _rt1, _rt2, _rt3, _rt4, _rt5, _rt6, _rt7 : R_TRIG;
    _w1, _w2 : BOOL;
    _ft1 : F_TRIG;
END_VAR

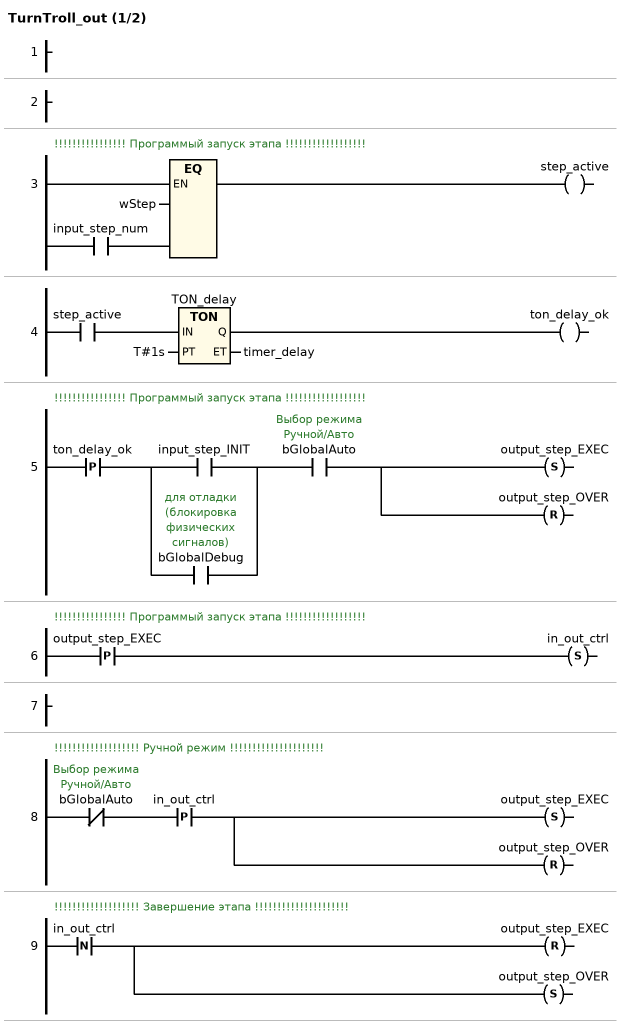
// NETWORK 1

// NETWORK 2

// NETWORK 3
// !!!!!!!!!!!!!!!! Программый запуск этапа !!!!!!!!!!!!!!!!!!
step_active := wStep = input_step_num;

// NETWORK 4
TON_delay(IN := step_active, PT := T#1s, ET => timer_delay); // TON
ton_delay_ok := TON_delay.Q;

// NETWORK 5
// !!!!!!!!!!!!!!!! Программый запуск этапа !!!!!!!!!!!!!!!!!!
//   bGlobalDebug: для отладки (блокировка физических сигналов)
//   bGlobalAuto: Выбор режима Ручной/Авто
_rt1(CLK := ton_delay_ok);
_w1 := _rt1.Q AND (input_step_INIT OR bGlobalDebug) AND bGlobalAuto;
output_step_EXEC S= _w1;
output_step_OVER R= _w1;

// NETWORK 6
// !!!!!!!!!!!!!!!! Программый запуск этапа !!!!!!!!!!!!!!!!!!
_rt2(CLK := output_step_EXEC);
in_out_ctrl S= _rt2.Q;

// NETWORK 7

// NETWORK 8
// !!!!!!!!!!!!!!!!!!! Ручной режим !!!!!!!!!!!!!!!!!!!!!
//   bGlobalAuto: Выбор режима Ручной/Авто
_rt3(CLK := in_out_ctrl);
_w2 := NOT bGlobalAuto AND _rt3.Q;
output_step_EXEC S= _w2;
output_step_OVER R= _w2;

// NETWORK 9
// !!!!!!!!!!!!!!!!!!! Завершение этапа !!!!!!!!!!!!!!!!!!!!!
_ft1(CLK := in_out_ctrl);
output_step_EXEC R= _ft1.Q;
output_step_OVER S= _ft1.Q;

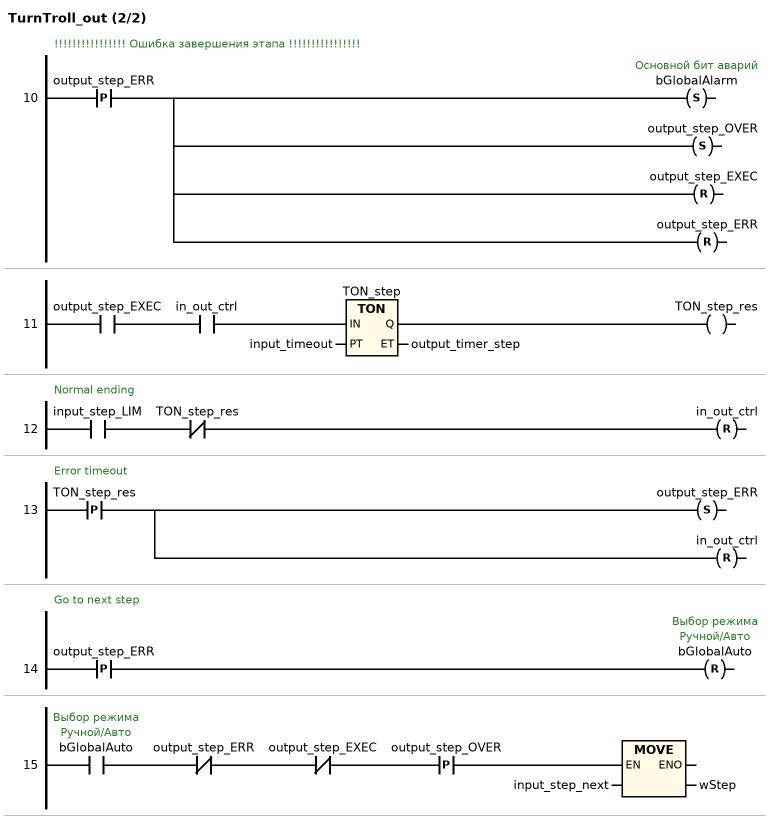
// NETWORK 10
// !!!!!!!!!!!!!!!! Ошибка завершения этапа !!!!!!!!!!!!!!!!
//   bGlobalAlarm: Основной бит аварий
_rt4(CLK := output_step_ERR);
bGlobalAlarm S= _rt4.Q;
output_step_OVER S= _rt4.Q;
output_step_EXEC R= _rt4.Q;
output_step_ERR R= _rt4.Q;

// NETWORK 11
TON_step(IN := output_step_EXEC AND in_out_ctrl, PT := input_timeout, ET => output_timer_step); // TON
TON_step_res := TON_step.Q;

// NETWORK 12
// Normal ending
in_out_ctrl R= input_step_LIM AND NOT TON_step_res;

// NETWORK 13
// Error timeout
_rt5(CLK := TON_step_res);
output_step_ERR S= _rt5.Q;
in_out_ctrl R= _rt5.Q;

// NETWORK 14
// Go to next step
//   bGlobalAuto: Выбор режима Ручной/Авто
_rt6(CLK := output_step_ERR);
bGlobalAuto R= _rt6.Q;

// NETWORK 15
//   bGlobalAuto: Выбор режима Ручной/Авто
_rt7(CLK := output_step_OVER);
IF bGlobalAuto AND NOT output_step_ERR AND NOT output_step_EXEC AND _rt7.Q THEN wStep := input_step_next; END_IF

END_PROGRAM

// MyController/Application/POU_6_HorizontalCutting
PROGRAM POU_6_HorizontalCutting
VAR
	step_MovingFrame_INIT: BOOL;
	sens_MovingFrame_fwd: BOOL;
	step_MovingFrame_fwd_EXEC: BOOL;
	step_MovingFrame_fwd_OVER: BOOL;
	step_MovingFrame_fwd_ERR: BOOL;
	timer_MovingFrame_fwd: TIME;
	sens_MovingFrame_rev: BOOL;
	step_MovingFrame_rev_EXEC: BOOL;
	step_MovingFrame_rev_OVER: BOOL;
	step_MovingFrame_rev_ERR: BOOL;
	timer_MovingFrame_rev: TIME;
END_VAR
VAR // added by the converter: edge detectors and wires of the graphical bodies
    _rt1, _rt2 : R_TRIG;
    _ft1, _ft2 : F_TRIG;
END_VAR

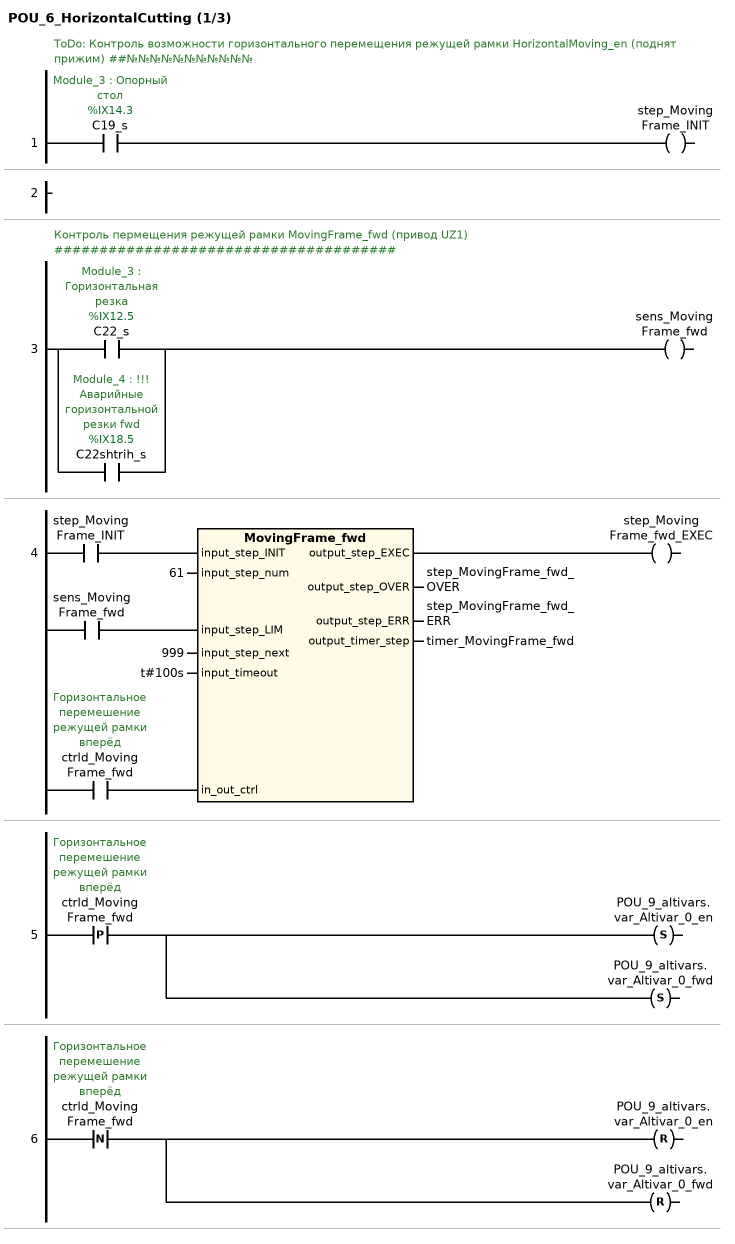
// NETWORK 1
// ToDo: Контроль возможности горизонтального перемещения режущей рамки HorizontalMoving_en (поднят прижим) ##№№№№№№№№№№№
//   C19_s: Module_3 : Опорный стол | AT %IX14.3
step_MovingFrame_INIT := C19_s;

// NETWORK 2

// NETWORK 3
// Контроль пермещения режущей рамки MovingFrame_fwd (привод UZ1) ######################################
//   C22_s: Module_3 : Горизонтальная резка | AT %IX12.5
//   C22shtrih_s: Module_4 : !!! Аварийные горизонтальной резки fwd | AT %IX18.5
sens_MovingFrame_fwd := C22_s OR C22shtrih_s;

// NETWORK 4
//   ctrld_MovingFrame_fwd: Горизонтальное перемешение режущей рамки вперёд
MovingFrame_fwd(input_step_INIT := step_MovingFrame_INIT, input_step_num := 61, input_step_LIM := sens_MovingFrame_fwd, input_step_next := 999, input_timeout := t#100s, in_out_ctrl := ctrld_MovingFrame_fwd, output_step_OVER => step_MovingFrame_fwd_OVER, output_step_ERR => step_MovingFrame_fwd_ERR, output_timer_step => timer_MovingFrame_fwd);
step_MovingFrame_fwd_EXEC := MovingFrame_fwd.output_step_EXEC;

// NETWORK 5
//   ctrld_MovingFrame_fwd: Горизонтальное перемешение режущей рамки вперёд
_rt1(CLK := ctrld_MovingFrame_fwd);
POU_9_altivars.var_Altivar_0_en S= _rt1.Q;
POU_9_altivars.var_Altivar_0_fwd S= _rt1.Q;

// NETWORK 6
//   ctrld_MovingFrame_fwd: Горизонтальное перемешение режущей рамки вперёд
_ft1(CLK := ctrld_MovingFrame_fwd);
POU_9_altivars.var_Altivar_0_en R= _ft1.Q;
POU_9_altivars.var_Altivar_0_fwd R= _ft1.Q;

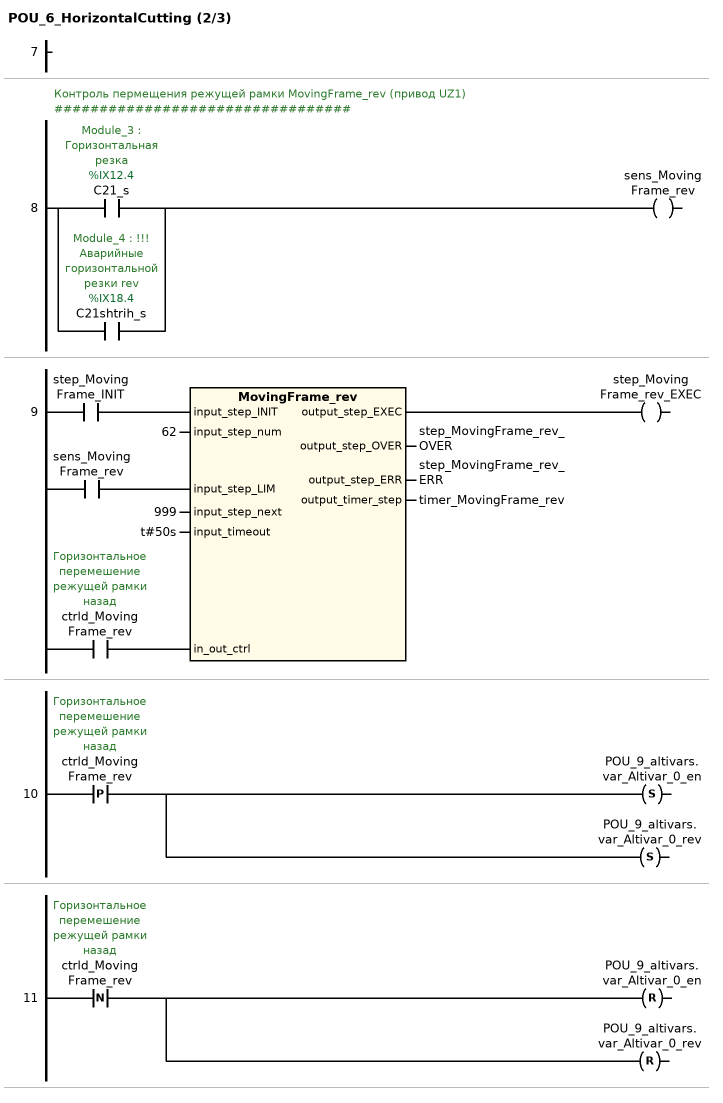
// NETWORK 7

// NETWORK 8
// Контроль пермещения режущей рамки MovingFrame_rev (привод UZ1) #################################
//   C21_s: Module_3 : Горизонтальная резка | AT %IX12.4
//   C21shtrih_s: Module_4 : !!! Аварийные горизонтальной резки rev | AT %IX18.4
sens_MovingFrame_rev := C21_s OR C21shtrih_s;

// NETWORK 9
//   ctrld_MovingFrame_rev: Горизонтальное перемешение режущей рамки назад
MovingFrame_rev(input_step_INIT := step_MovingFrame_INIT, input_step_num := 62, input_step_LIM := sens_MovingFrame_rev, input_step_next := 999, input_timeout := t#50s, in_out_ctrl := ctrld_MovingFrame_rev, output_step_OVER => step_MovingFrame_rev_OVER, output_step_ERR => step_MovingFrame_rev_ERR, output_timer_step => timer_MovingFrame_rev);
step_MovingFrame_rev_EXEC := MovingFrame_rev.output_step_EXEC;

// NETWORK 10
//   ctrld_MovingFrame_rev: Горизонтальное перемешение режущей рамки назад
_rt2(CLK := ctrld_MovingFrame_rev);
POU_9_altivars.var_Altivar_0_en S= _rt2.Q;
POU_9_altivars.var_Altivar_0_rev S= _rt2.Q;

// NETWORK 11
//   ctrld_MovingFrame_rev: Горизонтальное перемешение режущей рамки назад
_ft2(CLK := ctrld_MovingFrame_rev);
POU_9_altivars.var_Altivar_0_en R= _ft2.Q;
POU_9_altivars.var_Altivar_0_rev R= _ft2.Q;

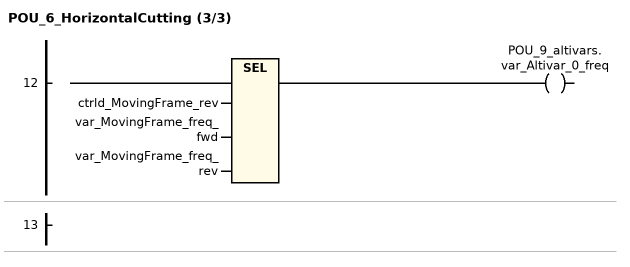
// NETWORK 12
//   ctrld_MovingFrame_rev: Горизонтальное перемешение режущей рамки назад
POU_9_altivars.var_Altivar_0_freq := SEL(ctrld_MovingFrame_rev, var_MovingFrame_freq_fwd, var_MovingFrame_freq_rev);

// NETWORK 13

END_PROGRAM

// MyController/Application/module_unites/MovingFrame_fwd
PROGRAM MovingFrame_fwd
VAR_INPUT
	input_step_INIT: BOOL;
	input_step_num: INT;
	input_step_LIM: BOOL;
	input_step_next: INT;
	input_timeout: TIME;
END_VAR

VAR_OUTPUT
	output_step_EXEC: BOOL;
	output_step_OVER: BOOL;
	output_step_ERR: BOOL;
	output_timer_step: TIME;
END_VAR
VAR_IN_OUT
	in_out_ctrl: BOOL;
END_VAR
VAR
	TON_step: TON;
	TON_step_res: BOOL;
	step_active: BOOL;
	TON_delay: TON;
	timer_delay: TIME;
	ton_delay_ok: BOOL;
END_VAR
VAR // added by the converter: edge detectors and wires of the graphical bodies
    _rt1, _rt2, _rt3, _rt4, _rt5, _rt6, _rt7 : R_TRIG;
    _w1, _w2 : BOOL;
    _ft1 : F_TRIG;
END_VAR

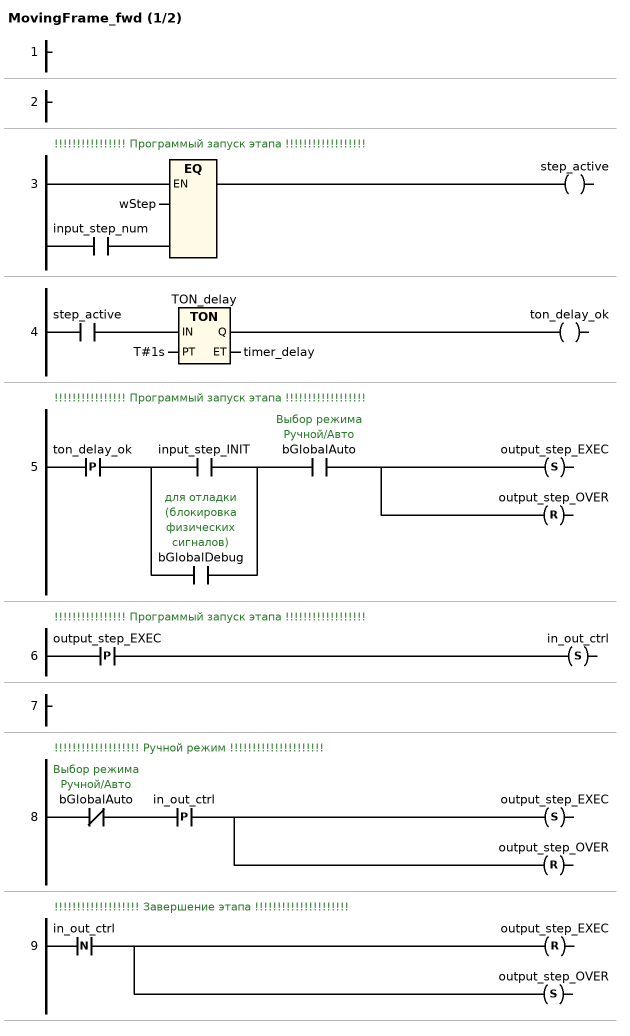
// NETWORK 1

// NETWORK 2

// NETWORK 3
// !!!!!!!!!!!!!!!! Программый запуск этапа !!!!!!!!!!!!!!!!!!
step_active := wStep = input_step_num;

// NETWORK 4
TON_delay(IN := step_active, PT := T#1s, ET => timer_delay); // TON
ton_delay_ok := TON_delay.Q;

// NETWORK 5
// !!!!!!!!!!!!!!!! Программый запуск этапа !!!!!!!!!!!!!!!!!!
//   bGlobalDebug: для отладки (блокировка физических сигналов)
//   bGlobalAuto: Выбор режима Ручной/Авто
_rt1(CLK := ton_delay_ok);
_w1 := _rt1.Q AND (input_step_INIT OR bGlobalDebug) AND bGlobalAuto;
output_step_EXEC S= _w1;
output_step_OVER R= _w1;

// NETWORK 6
// !!!!!!!!!!!!!!!! Программый запуск этапа !!!!!!!!!!!!!!!!!!
_rt2(CLK := output_step_EXEC);
in_out_ctrl S= _rt2.Q;

// NETWORK 7

// NETWORK 8
// !!!!!!!!!!!!!!!!!!! Ручной режим !!!!!!!!!!!!!!!!!!!!!
//   bGlobalAuto: Выбор режима Ручной/Авто
_rt3(CLK := in_out_ctrl);
_w2 := NOT bGlobalAuto AND _rt3.Q;
output_step_EXEC S= _w2;
output_step_OVER R= _w2;

// NETWORK 9
// !!!!!!!!!!!!!!!!!!! Завершение этапа !!!!!!!!!!!!!!!!!!!!!
_ft1(CLK := in_out_ctrl);
output_step_EXEC R= _ft1.Q;
output_step_OVER S= _ft1.Q;

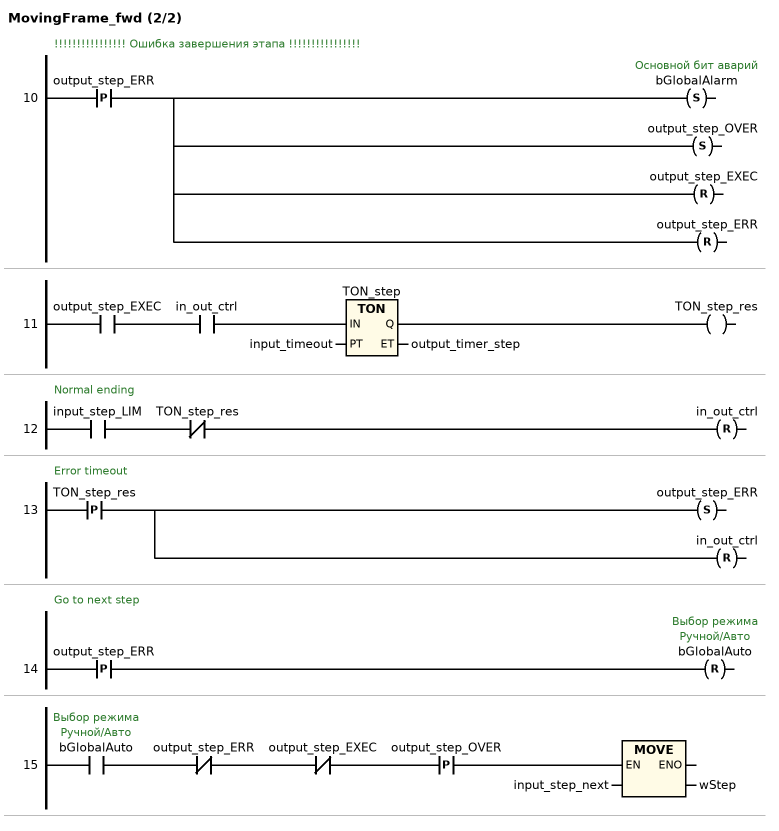
// NETWORK 10
// !!!!!!!!!!!!!!!! Ошибка завершения этапа !!!!!!!!!!!!!!!!
//   bGlobalAlarm: Основной бит аварий
_rt4(CLK := output_step_ERR);
bGlobalAlarm S= _rt4.Q;
output_step_OVER S= _rt4.Q;
output_step_EXEC R= _rt4.Q;
output_step_ERR R= _rt4.Q;

// NETWORK 11
TON_step(IN := output_step_EXEC AND in_out_ctrl, PT := input_timeout, ET => output_timer_step); // TON
TON_step_res := TON_step.Q;

// NETWORK 12
// Normal ending
in_out_ctrl R= input_step_LIM AND NOT TON_step_res;

// NETWORK 13
// Error timeout
_rt5(CLK := TON_step_res);
output_step_ERR S= _rt5.Q;
in_out_ctrl R= _rt5.Q;

// NETWORK 14
// Go to next step
//   bGlobalAuto: Выбор режима Ручной/Авто
_rt6(CLK := output_step_ERR);
bGlobalAuto R= _rt6.Q;

// NETWORK 15
//   bGlobalAuto: Выбор режима Ручной/Авто
_rt7(CLK := output_step_OVER);
IF bGlobalAuto AND NOT output_step_ERR AND NOT output_step_EXEC AND _rt7.Q THEN wStep := input_step_next; END_IF

END_PROGRAM

// MyController/Application/module_unites/MovingFrame_rev
PROGRAM MovingFrame_rev
VAR_INPUT
	input_step_INIT: BOOL;
	input_step_num: INT;
	input_step_LIM: BOOL;
	input_step_next: INT;
	input_timeout: TIME;
END_VAR

VAR_OUTPUT
	output_step_EXEC: BOOL;
	output_step_OVER: BOOL;
	output_step_ERR: BOOL;
	output_timer_step: TIME;
END_VAR
VAR_IN_OUT
	in_out_ctrl: BOOL;
END_VAR
VAR
	TON_step: TON;
	TON_step_res: BOOL;
	step_active: BOOL;
	TON_delay: TON;
	timer_delay: TIME;
	ton_delay_ok: BOOL;
END_VAR
VAR // added by the converter: edge detectors and wires of the graphical bodies
    _rt1, _rt2, _rt3, _rt4, _rt5, _rt6, _rt7 : R_TRIG;
    _w1, _w2 : BOOL;
    _ft1 : F_TRIG;
END_VAR

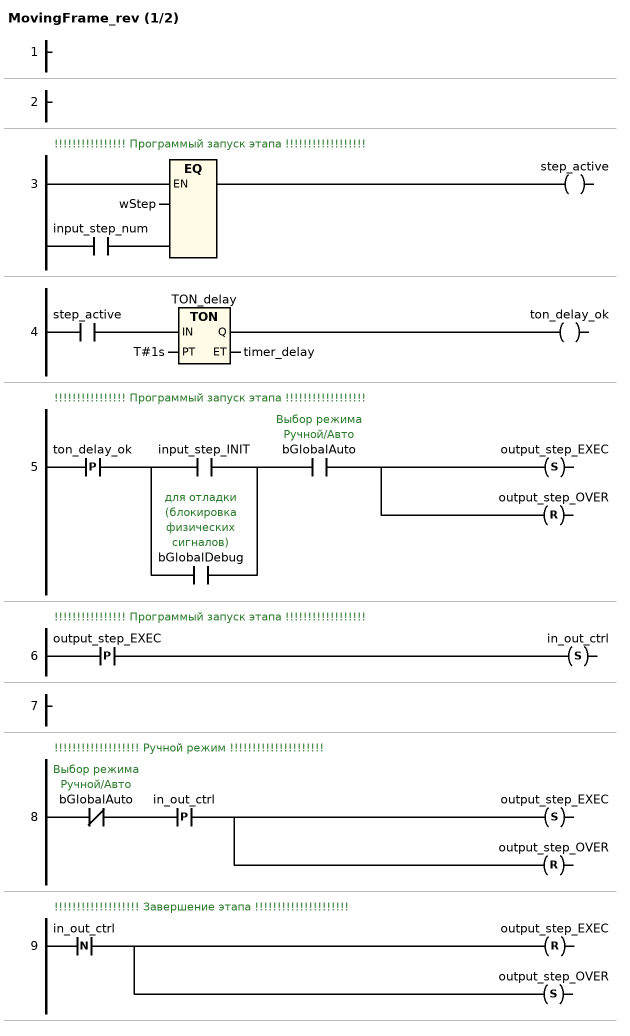
// NETWORK 1

// NETWORK 2

// NETWORK 3
// !!!!!!!!!!!!!!!! Программый запуск этапа !!!!!!!!!!!!!!!!!!
step_active := wStep = input_step_num;

// NETWORK 4
TON_delay(IN := step_active, PT := T#1s, ET => timer_delay); // TON
ton_delay_ok := TON_delay.Q;

// NETWORK 5
// !!!!!!!!!!!!!!!! Программый запуск этапа !!!!!!!!!!!!!!!!!!
//   bGlobalDebug: для отладки (блокировка физических сигналов)
//   bGlobalAuto: Выбор режима Ручной/Авто
_rt1(CLK := ton_delay_ok);
_w1 := _rt1.Q AND (input_step_INIT OR bGlobalDebug) AND bGlobalAuto;
output_step_EXEC S= _w1;
output_step_OVER R= _w1;

// NETWORK 6
// !!!!!!!!!!!!!!!! Программый запуск этапа !!!!!!!!!!!!!!!!!!
_rt2(CLK := output_step_EXEC);
in_out_ctrl S= _rt2.Q;

// NETWORK 7

// NETWORK 8
// !!!!!!!!!!!!!!!!!!! Ручной режим !!!!!!!!!!!!!!!!!!!!!
//   bGlobalAuto: Выбор режима Ручной/Авто
_rt3(CLK := in_out_ctrl);
_w2 := NOT bGlobalAuto AND _rt3.Q;
output_step_EXEC S= _w2;
output_step_OVER R= _w2;

// NETWORK 9
// !!!!!!!!!!!!!!!!!!! Завершение этапа !!!!!!!!!!!!!!!!!!!!!
_ft1(CLK := in_out_ctrl);
output_step_EXEC R= _ft1.Q;
output_step_OVER S= _ft1.Q;

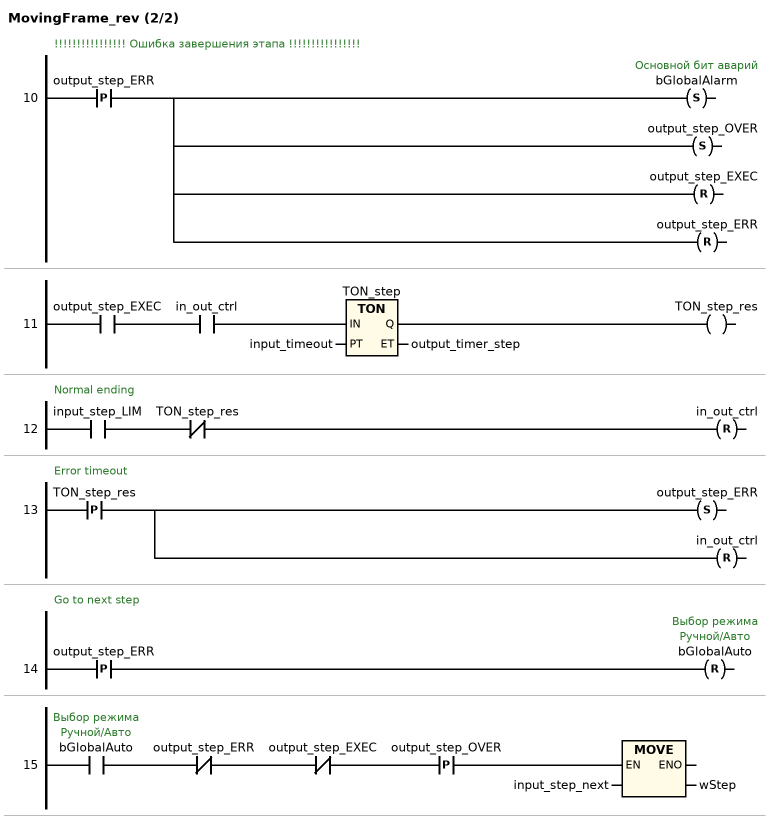
// NETWORK 10
// !!!!!!!!!!!!!!!! Ошибка завершения этапа !!!!!!!!!!!!!!!!
//   bGlobalAlarm: Основной бит аварий
_rt4(CLK := output_step_ERR);
bGlobalAlarm S= _rt4.Q;
output_step_OVER S= _rt4.Q;
output_step_EXEC R= _rt4.Q;
output_step_ERR R= _rt4.Q;

// NETWORK 11
TON_step(IN := output_step_EXEC AND in_out_ctrl, PT := input_timeout, ET => output_timer_step); // TON
TON_step_res := TON_step.Q;

// NETWORK 12
// Normal ending
in_out_ctrl R= input_step_LIM AND NOT TON_step_res;

// NETWORK 13
// Error timeout
_rt5(CLK := TON_step_res);
output_step_ERR S= _rt5.Q;
in_out_ctrl R= _rt5.Q;

// NETWORK 14
// Go to next step
//   bGlobalAuto: Выбор режима Ручной/Авто
_rt6(CLK := output_step_ERR);
bGlobalAuto R= _rt6.Q;

// NETWORK 15
//   bGlobalAuto: Выбор режима Ручной/Авто
_rt7(CLK := output_step_OVER);
IF bGlobalAuto AND NOT output_step_ERR AND NOT output_step_EXEC AND _rt7.Q THEN wStep := input_step_next; END_IF

END_PROGRAM

// MyController/Application/POU_7_VerticalCutting
PROGRAM POU_7_VerticalCutting
VAR
	step_PressTable_INIT: BOOL := TRUE;
	ctrl_PressTable_in: BOOL;
	sens_PressTable_in: BOOL;
	step_PressTable_in_EXEC: BOOL;
	step_PressTable_in_OVER: BOOL;
	step_PressTable_in_ERR: BOOL;
	timer_PressTable_in: TIME;
	timer_PressTable_out: TIME;
	ctrl_PressTable_out: BOOL;
	sens_PressTable_out: BOOL;
	step_PressTable_out_EXEC: BOOL;
	step_PressTable_out_OVER: BOOL;
	step_PressTable_out_ERR: BOOL;
	sens_CuttingFrame_up: BOOL;
	sens_CuttingFrame_dn: BOOL;
	step_CuttingFrame_INIT: BOOL := TRUE;
	step_CuttingFrame_in_EXEC: BOOL;
	step_CuttingFrame_up_OVER: BOOL;
	step_CuttingFrame_up_EXEC: BOOL;
	step_CuttingFrame_up_ERR: BOOL;
	timer_CuttingFrame_up: TIME;
	step_CuttingFrame_dn_EXEC: BOOL;
	step_CuttingFrame_dn_OVER: BOOL;
	step_CuttingFrame_dn_ERR: BOOL;
	timer_CuttingFrame_dn: TIME;
END_VAR
VAR // added by the converter: edge detectors and wires of the graphical bodies
    _rt1, _rt2 : R_TRIG;
    _ft1, _ft2 : F_TRIG;
END_VAR

